{attribute 'qualified_only'}
{attribute 'strict'}
TYPE E_CSL_Colors :
(
	
	
);
END_TYPE

(* stored: Version 1.1.0.1, ProductVersion 3.1.4024.12
   EnumerationTextList E_CSL_Colors: Id {6f1ef125-03be-4339-962f-6a12e66182b8} *)
